// LS Electric XG5000 project: Dois_Inversores_S100_Ethernet
// PLC Main

PROGRAM Comandos (task: Scan Program)

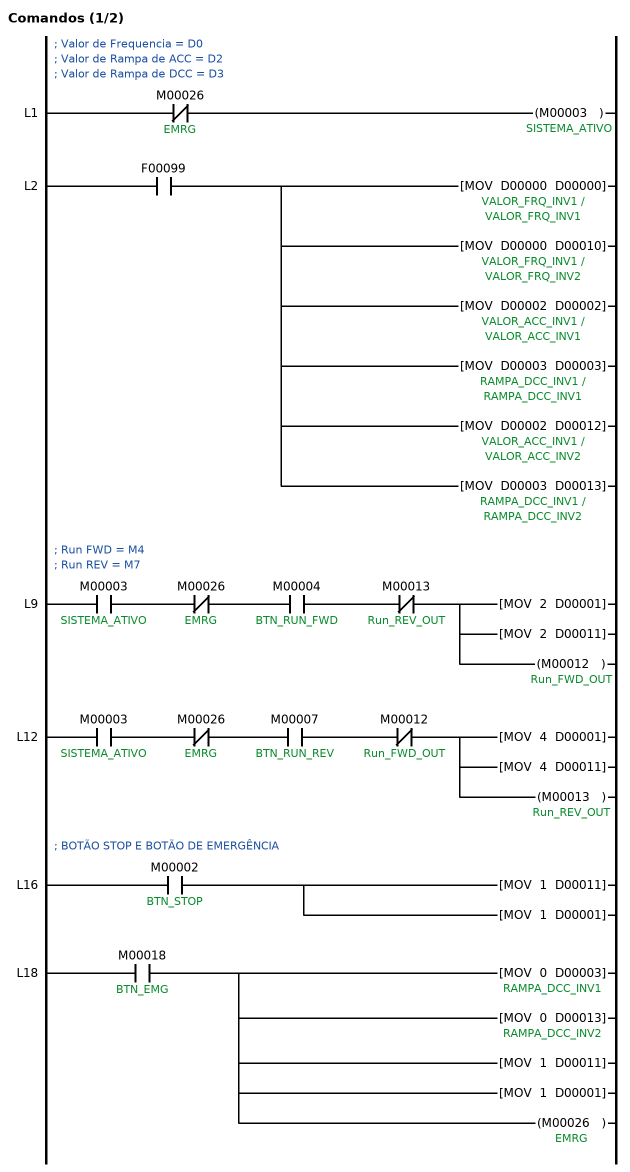
// Valor de Frequencia = D0
// Valor de Rampa de ACC = D2
// Valor de Rampa de DCC = D3
; L1
LOAD NOT  M00026	// EMRG
OUT       M00003	// SISTEMA_ATIVO
; L2
LOAD      F00099
MOV       D00000 D00000	// VALOR_FRQ_INV1 / VALOR_FRQ_INV1
MOV       D00000 D00010	// VALOR_FRQ_INV1 / VALOR_FRQ_INV2
MOV       D00002 D00002	// VALOR_ACC_INV1 / VALOR_ACC_INV1
MOV       D00003 D00003	// RAMPA_DCC_INV1 / RAMPA_DCC_INV1
MOV       D00002 D00012	// VALOR_ACC_INV1 / VALOR_ACC_INV2
MOV       D00003 D00013	// RAMPA_DCC_INV1 / RAMPA_DCC_INV2
// Run FWD = M4
// Run REV = M7
; L9
LOAD      M00003	// SISTEMA_ATIVO
AND NOT   M00026	// EMRG
AND       M00004	// BTN_RUN_FWD
AND NOT   M00013	// Run_REV_OUT
MOV       2 D00001
MOV       2 D00011
OUT       M00012	// Run_FWD_OUT
; L12
LOAD      M00003	// SISTEMA_ATIVO
AND NOT   M00026	// EMRG
AND       M00007	// BTN_RUN_REV
AND NOT   M00012	// Run_FWD_OUT
MOV       4 D00001
MOV       4 D00011
OUT       M00013	// Run_REV_OUT
// BOTÃO STOP E BOTÃO DE EMERGÊNCIA
; L16
LOAD      M00002	// BTN_STOP
MOV       1 D00011
MOV       1 D00001
; L18
LOAD      M00018	// BTN_EMG
MOV       0 D00003	// RAMPA_DCC_INV1
MOV       0 D00013	// RAMPA_DCC_INV2
MOV       1 D00011
MOV       1 D00001
OUT       M00026	// EMRG

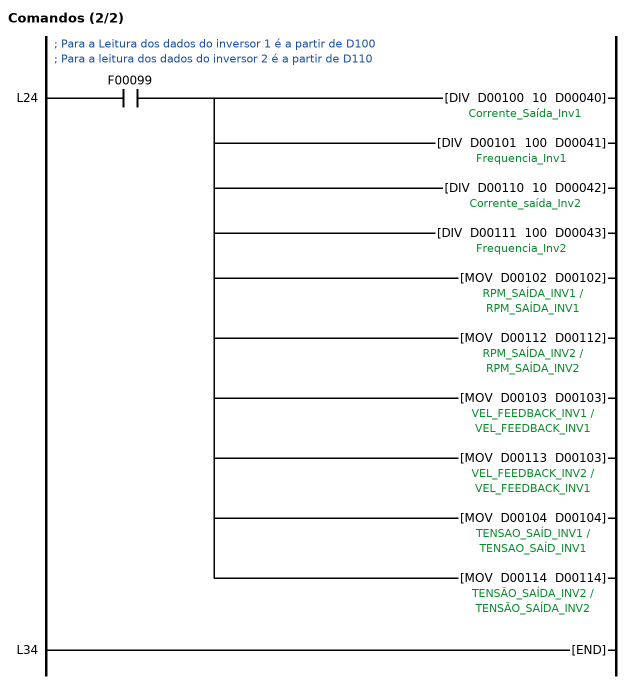
// Para a Leitura dos dados do inversor 1 é a partir de D100
// Para a leitura dos dados do inversor 2 é a partir de D110
; L24
LOAD      F00099
DIV       D00100 10 D00040	// Corrente_Saída_Inv1
DIV       D00101 100 D00041	// Frequencia_Inv1
DIV       D00110 10 D00042	// Corrente_saída_Inv2
DIV       D00111 100 D00043	// Frequencia_Inv2
MOV       D00102 D00102	// RPM_SAÍDA_INV1 / RPM_SAÍDA_INV1
MOV       D00112 D00112	// RPM_SAÍDA_INV2 / RPM_SAÍDA_INV2
MOV       D00103 D00103	// VEL_FEEDBACK_INV1 / VEL_FEEDBACK_INV1
MOV       D00113 D00103	// VEL_FEEDBACK_INV2 / VEL_FEEDBACK_INV1
MOV       D00104 D00104	// TENSAO_SAÍD_INV1 / TENSAO_SAÍD_INV1
MOV       D00114 D00114	// TENSÃO_SAÍDA_INV2 / TENSÃO_SAÍDA_INV2
; L34
END

VARIABLES AND COMMENTS (devices not used above)
M00005	BIT	MOTOR_REV
M00001	BIT	Run_FWD
M00006	BIT	RUN_REV
M00025	BIT	STOP